PROGRAM PRG_05_Turret_Carriage
VAR
	R_TRIG_0: R_TRIG;
	R_TRIG_1: R_TRIG;
	F_TRIG_2: F_TRIG;
	F_TRIG_4: F_TRIG;
	RS_TriggerStopCCW: RS;
	R_TRIG_12: R_TRIG;
	RS_TriggerStopCW: RS;
	R_TRIG_15: R_TRIG;
	R_TRIG_18: R_TRIG;
	R_TRIG_19: R_TRIG;
	R_TRIG_20: R_TRIG;
	R_TRIG_21: R_TRIG;
	R_TRIG_22: R_TRIG;
	TOF_SwitchDelay: TOF;
	R_TRIG_23: R_TRIG;
	R_TRIG_24: R_TRIG;
	R_TRIG_25: R_TRIG;
	R_TRIG_26: R_TRIG;
	F_TRIG_0: F_TRIG;
	F_TRIG_1: F_TRIG;
END_VAR
VAR // added by the converter: edge detectors and wires of the graphical bodies
    _w1, _w2 : BOOL;
END_VAR

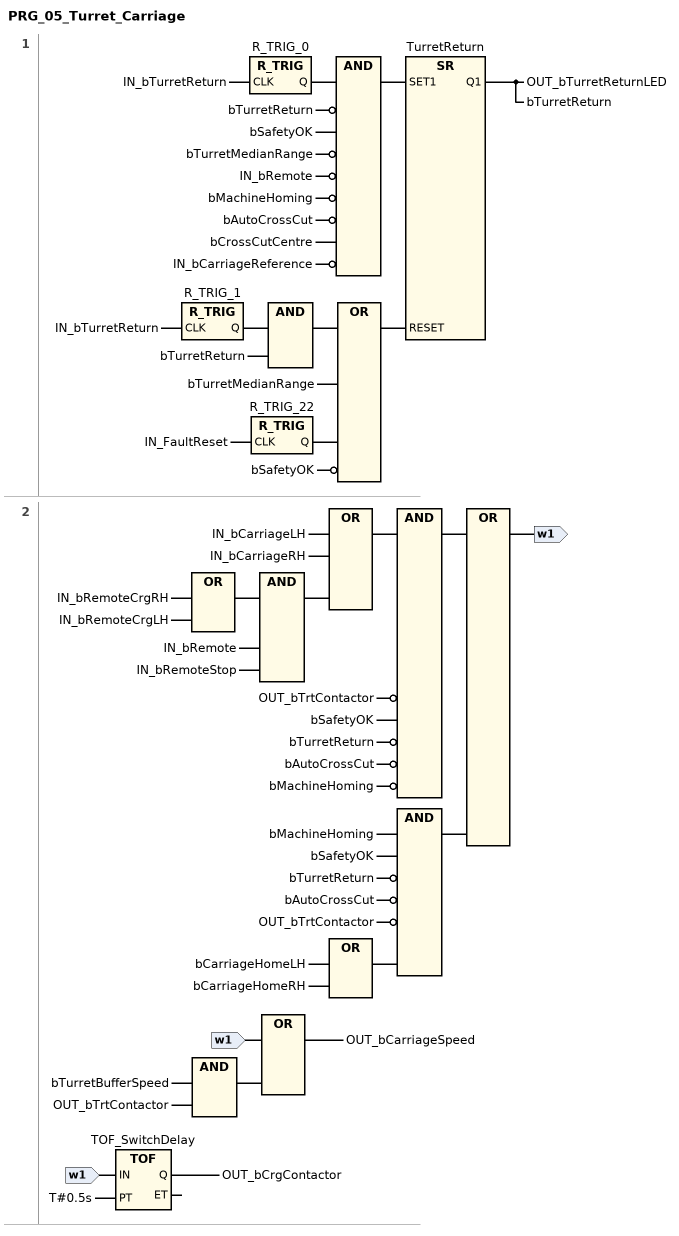
// NETWORK 1
R_TRIG_0(CLK := IN_bTurretReturn); // R_TRIG
R_TRIG_1(CLK := IN_bTurretReturn); // R_TRIG
R_TRIG_22(CLK := IN_FaultReset); // R_TRIG
TurretReturn(SET1 := R_TRIG_0.Q AND NOT bTurretReturn AND bSafetyOK AND NOT bTurretMedianRange AND NOT IN_bRemote AND NOT bMachineHoming AND NOT bAutoCrossCut AND bCrossCutCentre AND NOT IN_bCarriageReference, RESET := R_TRIG_1.Q AND bTurretReturn OR bTurretMedianRange OR R_TRIG_22.Q OR NOT bSafetyOK); // SR
OUT_bTurretReturnLED := TurretReturn.Q1;
bTurretReturn := TurretReturn.Q1;

// NETWORK 2
_w1 := (IN_bCarriageLH OR IN_bCarriageRH OR (IN_bRemoteCrgRH OR IN_bRemoteCrgLH) AND IN_bRemote AND IN_bRemoteStop) AND NOT OUT_bTrtContactor AND bSafetyOK AND NOT bTurretReturn AND NOT bAutoCrossCut AND NOT bMachineHoming OR bMachineHoming AND bSafetyOK AND NOT bTurretReturn AND NOT bAutoCrossCut AND NOT OUT_bTrtContactor AND (bCarriageHomeLH OR bCarriageHomeRH);
OUT_bCarriageSpeed := _w1 OR bTurretBufferSpeed AND OUT_bTrtContactor;
TOF_SwitchDelay(IN := _w1, PT := T#0.5s); // TOF
OUT_bCrgContactor := TOF_SwitchDelay.Q;

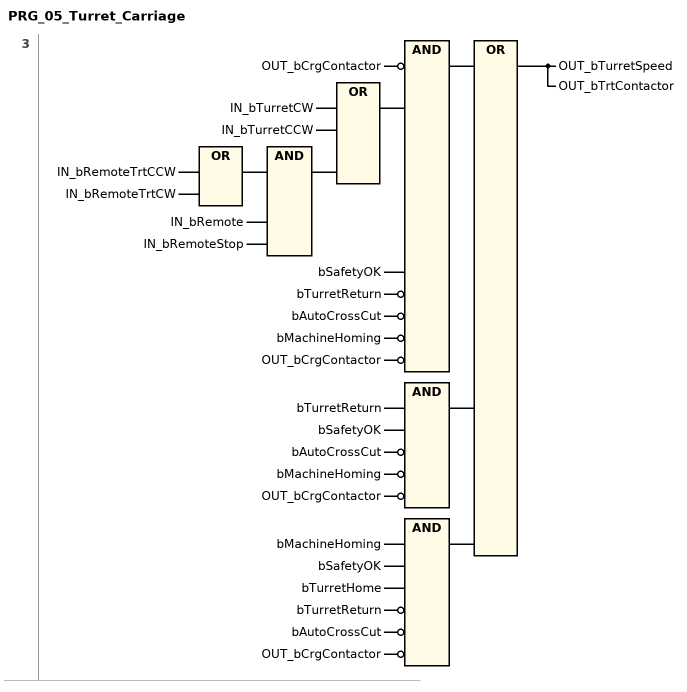
// NETWORK 3
_w2 := NOT OUT_bCrgContactor AND (IN_bTurretCW OR IN_bTurretCCW OR (IN_bRemoteTrtCCW OR IN_bRemoteTrtCW) AND IN_bRemote AND IN_bRemoteStop) AND bSafetyOK AND NOT bTurretReturn AND NOT bAutoCrossCut AND NOT bMachineHoming AND NOT OUT_bCrgContactor OR bTurretReturn AND bSafetyOK AND NOT bAutoCrossCut AND NOT bMachineHoming AND NOT OUT_bCrgContactor OR bMachineHoming AND bSafetyOK AND bTurretHome AND NOT bTurretReturn AND NOT bAutoCrossCut AND NOT OUT_bCrgContactor;
OUT_bTurretSpeed := _w2;
OUT_bTrtContactor := _w2;

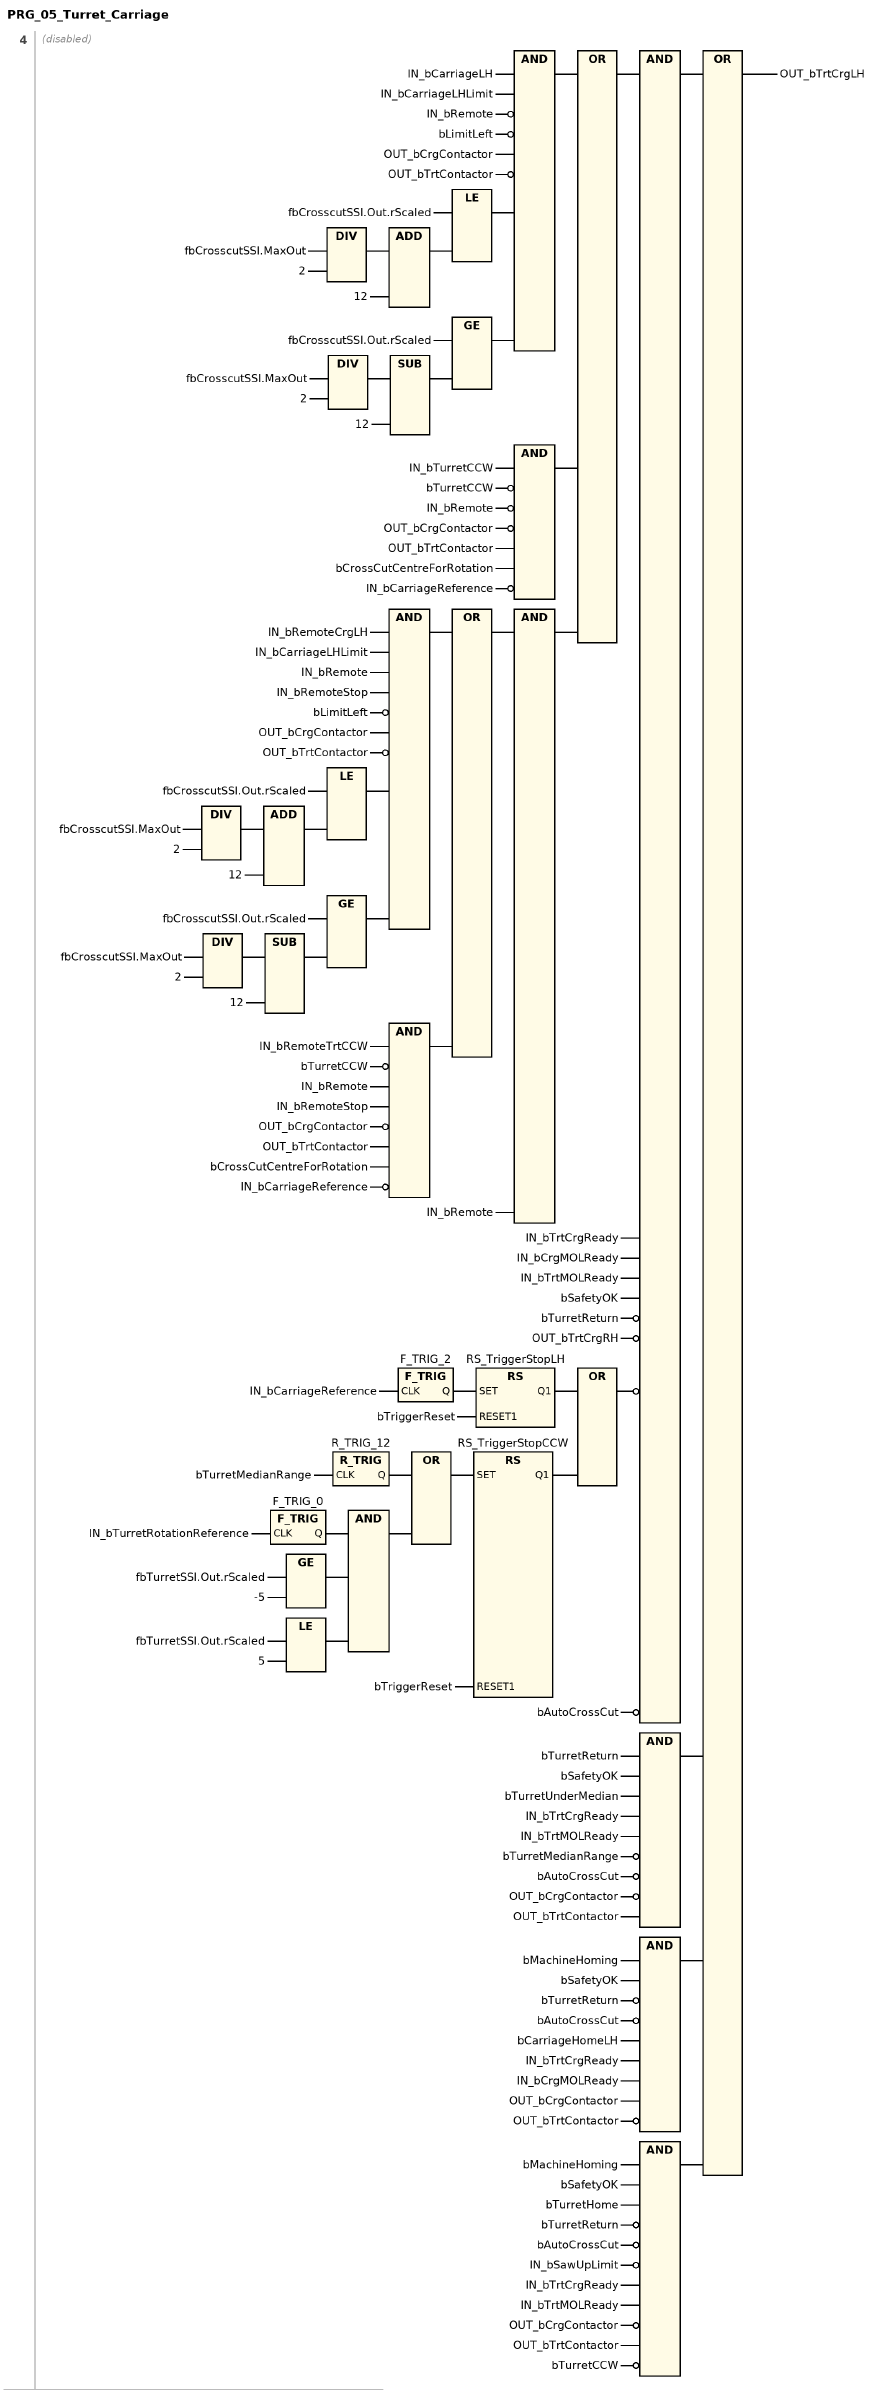
// NETWORK 4 (disabled)
// F_TRIG_2(CLK := IN_bCarriageReference); // F_TRIG
// RS_TriggerStopLH(SET := F_TRIG_2.Q, RESET1 := bTriggerReset); // RS
// R_TRIG_12(CLK := bTurretMedianRange); // R_TRIG
// F_TRIG_0(CLK := IN_bTurretRotationReference); // F_TRIG
// RS_TriggerStopCCW(SET := R_TRIG_12.Q OR F_TRIG_0.Q AND fbTurretSSI.Out.rScaled >= -5 AND fbTurretSSI.Out.rScaled <= 5, RESET1 := bTriggerReset); // RS
// OUT_bTrtCrgLH := (IN_bCarriageLH AND IN_bCarriageLHLimit AND NOT IN_bRemote AND NOT bLimitLeft AND OUT_bCrgContactor AND NOT OUT_bTrtContactor AND fbCrosscutSSI.Out.rScaled <= fbCrosscutSSI.MaxOut / 2 + 12 AND fbCrosscutSSI.Out.rScaled >= fbCrosscutSSI.MaxOut / 2 - 12 OR IN_bTurretCCW AND NOT bTurretCCW AND NOT IN_bRemote AND NOT OUT_bCrgContactor AND OUT_bTrtContactor AND bCrossCutCentreForRotation AND NOT IN_bCarriageReference OR (IN_bRemoteCrgLH AND IN_bCarriageLHLimit AND IN_bRemote AND IN_bRemoteStop AND NOT bLimitLeft AND OUT_bCrgContactor AND NOT OUT_bTrtContactor AND fbCrosscutSSI.Out.rScaled <= fbCrosscutSSI.MaxOut / 2 + 12 AND fbCrosscutSSI.Out.rScaled >= fbCrosscutSSI.MaxOut / 2 - 12 OR IN_bRemoteTrtCCW AND NOT bTurretCCW AND IN_bRemote AND IN_bRemoteStop AND NOT OUT_bCrgContactor AND OUT_bTrtContactor AND bCrossCutCentreForRotation AND NOT IN_bCarriageReference) AND IN_bRemote) AND IN_bTrtCrgReady AND IN_bCrgMOLReady AND IN_bTrtMOLReady AND bSafetyOK AND NOT bTurretReturn AND NOT OUT_bTrtCrgRH AND NOT (RS_TriggerStopLH.Q1 OR RS_TriggerStopCCW.Q1) AND NOT bAutoCrossCut OR bTurretReturn AND bSafetyOK AND bTurretUnderMedian AND IN_bTrtCrgReady AND IN_bTrtMOLReady AND NOT bTurretMedianRange AND NOT bAutoCrossCut AND NOT OUT_bCrgContactor AND OUT_bTrtContactor OR bMachineHoming AND bSafetyOK AND NOT bTurretReturn AND NOT bAutoCrossCut AND bCarriageHomeLH AND IN_bTrtCrgReady AND IN_bCrgMOLReady AND OUT_bCrgContactor AND NOT OUT_bTrtContactor OR bMachineHoming AND bSafetyOK AND bTurretHome AND NOT bTurretReturn AND NOT bAutoCrossCut AND NOT IN_bSawUpLimit AND IN_bTrtCrgReady AND IN_bTrtMOLReady AND NOT OUT_bCrgContactor AND OUT_bTrtContactor AND NOT bTurretCCW;

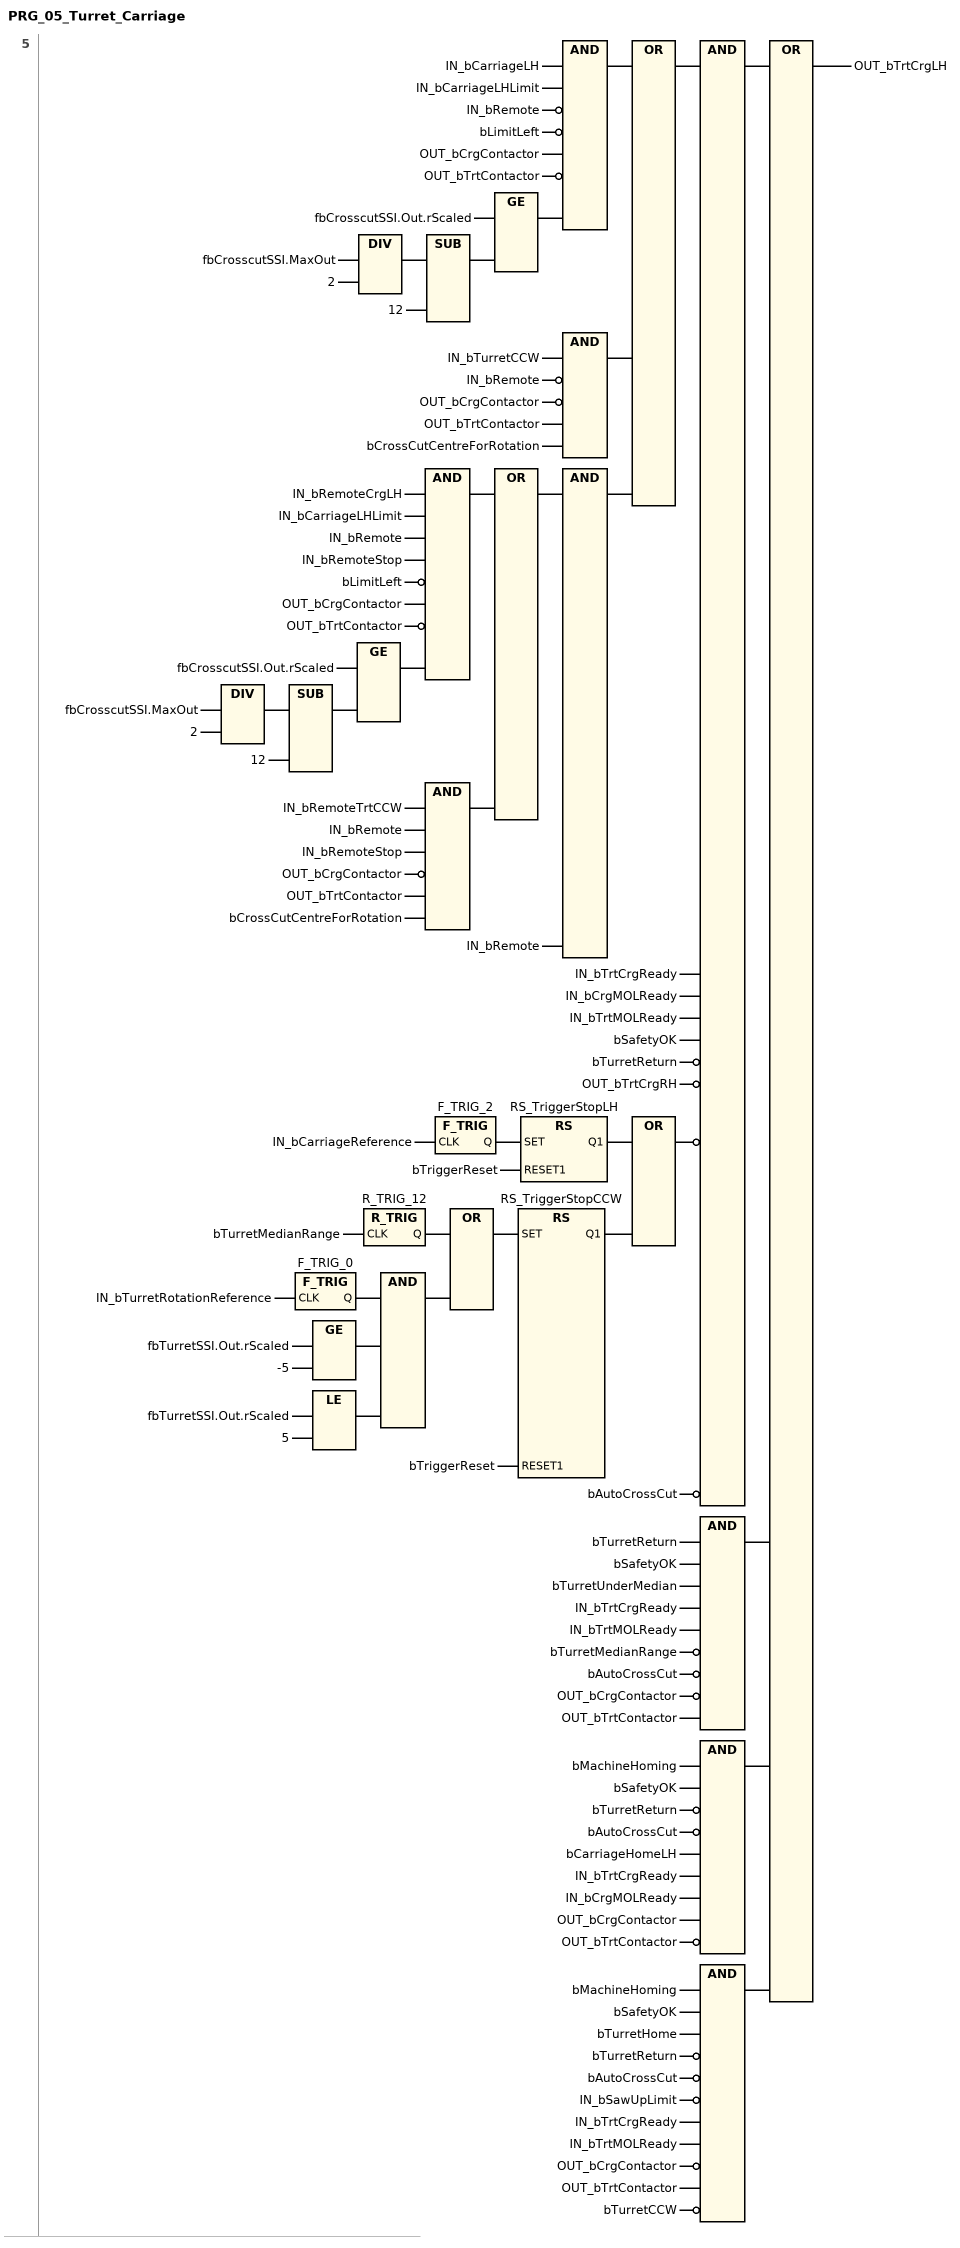
// NETWORK 5
F_TRIG_2(CLK := IN_bCarriageReference); // F_TRIG
RS_TriggerStopLH(SET := F_TRIG_2.Q, RESET1 := bTriggerReset); // RS
R_TRIG_12(CLK := bTurretMedianRange); // R_TRIG
F_TRIG_0(CLK := IN_bTurretRotationReference); // F_TRIG
RS_TriggerStopCCW(SET := R_TRIG_12.Q OR F_TRIG_0.Q AND fbTurretSSI.Out.rScaled >= -5 AND fbTurretSSI.Out.rScaled <= 5, RESET1 := bTriggerReset); // RS
OUT_bTrtCrgLH := (IN_bCarriageLH AND IN_bCarriageLHLimit AND NOT IN_bRemote AND NOT bLimitLeft AND OUT_bCrgContactor AND NOT OUT_bTrtContactor AND fbCrosscutSSI.Out.rScaled >= fbCrosscutSSI.MaxOut / 2 - 12 OR IN_bTurretCCW AND NOT IN_bRemote AND NOT OUT_bCrgContactor AND OUT_bTrtContactor AND bCrossCutCentreForRotation OR (IN_bRemoteCrgLH AND IN_bCarriageLHLimit AND IN_bRemote AND IN_bRemoteStop AND NOT bLimitLeft AND OUT_bCrgContactor AND NOT OUT_bTrtContactor AND fbCrosscutSSI.Out.rScaled >= fbCrosscutSSI.MaxOut / 2 - 12 OR IN_bRemoteTrtCCW AND IN_bRemote AND IN_bRemoteStop AND NOT OUT_bCrgContactor AND OUT_bTrtContactor AND bCrossCutCentreForRotation) AND IN_bRemote) AND IN_bTrtCrgReady AND IN_bCrgMOLReady AND IN_bTrtMOLReady AND bSafetyOK AND NOT bTurretReturn AND NOT OUT_bTrtCrgRH AND NOT (RS_TriggerStopLH.Q1 OR RS_TriggerStopCCW.Q1) AND NOT bAutoCrossCut OR bTurretReturn AND bSafetyOK AND bTurretUnderMedian AND IN_bTrtCrgReady AND IN_bTrtMOLReady AND NOT bTurretMedianRange AND NOT bAutoCrossCut AND NOT OUT_bCrgContactor AND OUT_bTrtContactor OR bMachineHoming AND bSafetyOK AND NOT bTurretReturn AND NOT bAutoCrossCut AND bCarriageHomeLH AND IN_bTrtCrgReady AND IN_bCrgMOLReady AND OUT_bCrgContactor AND NOT OUT_bTrtContactor OR bMachineHoming AND bSafetyOK AND bTurretHome AND NOT bTurretReturn AND NOT bAutoCrossCut AND NOT IN_bSawUpLimit AND IN_bTrtCrgReady AND IN_bTrtMOLReady AND NOT OUT_bCrgContactor AND OUT_bTrtContactor AND NOT bTurretCCW;

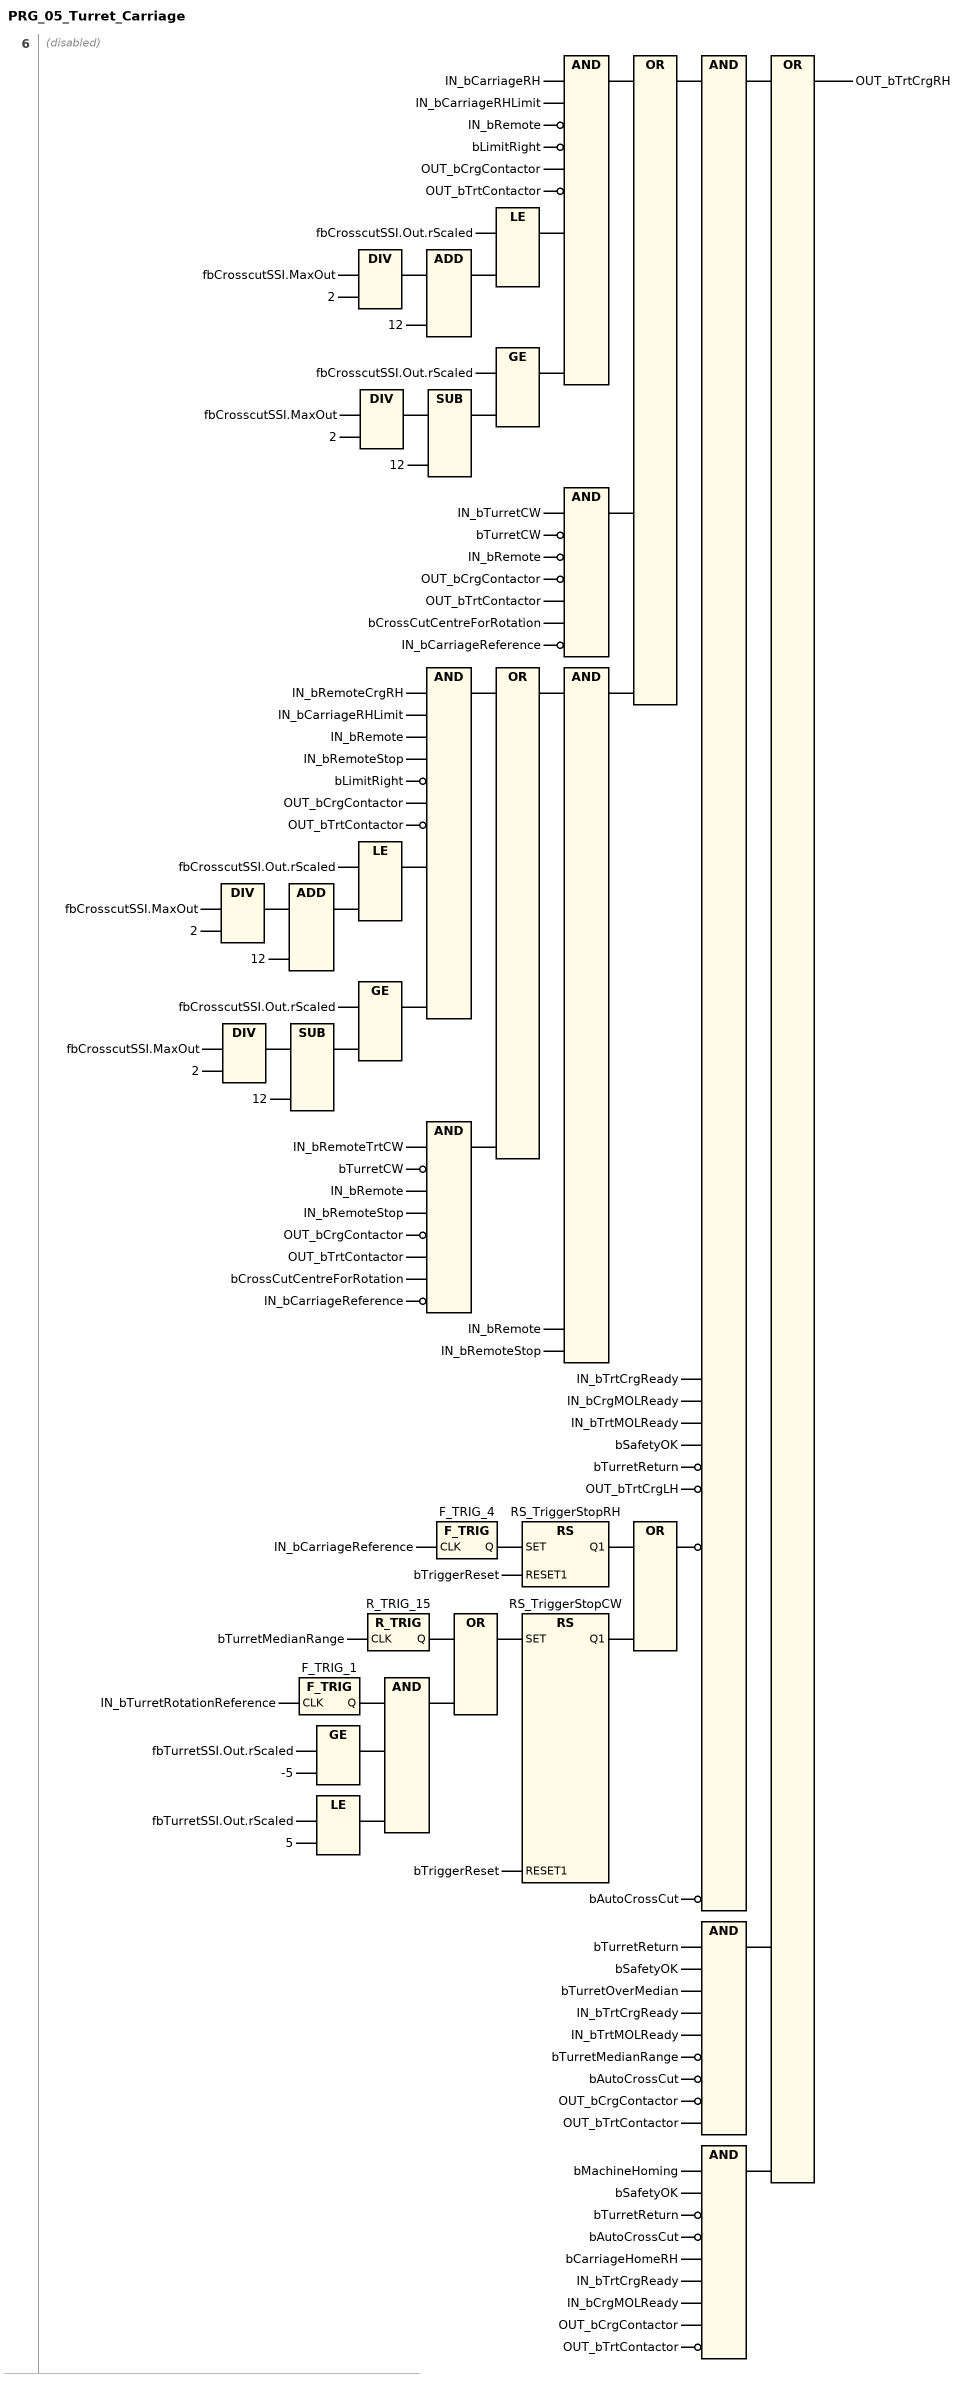
// NETWORK 6 (disabled)
// F_TRIG_4(CLK := IN_bCarriageReference); // F_TRIG
// RS_TriggerStopRH(SET := F_TRIG_4.Q, RESET1 := bTriggerReset); // RS
// R_TRIG_15(CLK := bTurretMedianRange); // R_TRIG
// F_TRIG_1(CLK := IN_bTurretRotationReference); // F_TRIG
// RS_TriggerStopCW(SET := R_TRIG_15.Q OR F_TRIG_1.Q AND fbTurretSSI.Out.rScaled >= -5 AND fbTurretSSI.Out.rScaled <= 5, RESET1 := bTriggerReset); // RS
// OUT_bTrtCrgRH := (IN_bCarriageRH AND IN_bCarriageRHLimit AND NOT IN_bRemote AND NOT bLimitRight AND OUT_bCrgContactor AND NOT OUT_bTrtContactor AND fbCrosscutSSI.Out.rScaled <= fbCrosscutSSI.MaxOut / 2 + 12 AND fbCrosscutSSI.Out.rScaled >= fbCrosscutSSI.MaxOut / 2 - 12 OR IN_bTurretCW AND NOT bTurretCW AND NOT IN_bRemote AND NOT OUT_bCrgContactor AND OUT_bTrtContactor AND bCrossCutCentreForRotation AND NOT IN_bCarriageReference OR (IN_bRemoteCrgRH AND IN_bCarriageRHLimit AND IN_bRemote AND IN_bRemoteStop AND NOT bLimitRight AND OUT_bCrgContactor AND NOT OUT_bTrtContactor AND fbCrosscutSSI.Out.rScaled <= fbCrosscutSSI.MaxOut / 2 + 12 AND fbCrosscutSSI.Out.rScaled >= fbCrosscutSSI.MaxOut / 2 - 12 OR IN_bRemoteTrtCW AND NOT bTurretCW AND IN_bRemote AND IN_bRemoteStop AND NOT OUT_bCrgContactor AND OUT_bTrtContactor AND bCrossCutCentreForRotation AND NOT IN_bCarriageReference) AND IN_bRemote AND IN_bRemoteStop) AND IN_bTrtCrgReady AND IN_bCrgMOLReady AND IN_bTrtMOLReady AND bSafetyOK AND NOT bTurretReturn AND NOT OUT_bTrtCrgLH AND NOT (RS_TriggerStopRH.Q1 OR RS_TriggerStopCW.Q1) AND NOT bAutoCrossCut OR bTurretReturn AND bSafetyOK AND bTurretOverMedian AND IN_bTrtCrgReady AND IN_bTrtMOLReady AND NOT bTurretMedianRange AND NOT bAutoCrossCut AND NOT OUT_bCrgContactor AND OUT_bTrtContactor OR bMachineHoming AND bSafetyOK AND NOT bTurretReturn AND NOT bAutoCrossCut AND bCarriageHomeRH AND IN_bTrtCrgReady AND IN_bCrgMOLReady AND OUT_bCrgContactor AND NOT OUT_bTrtContactor;

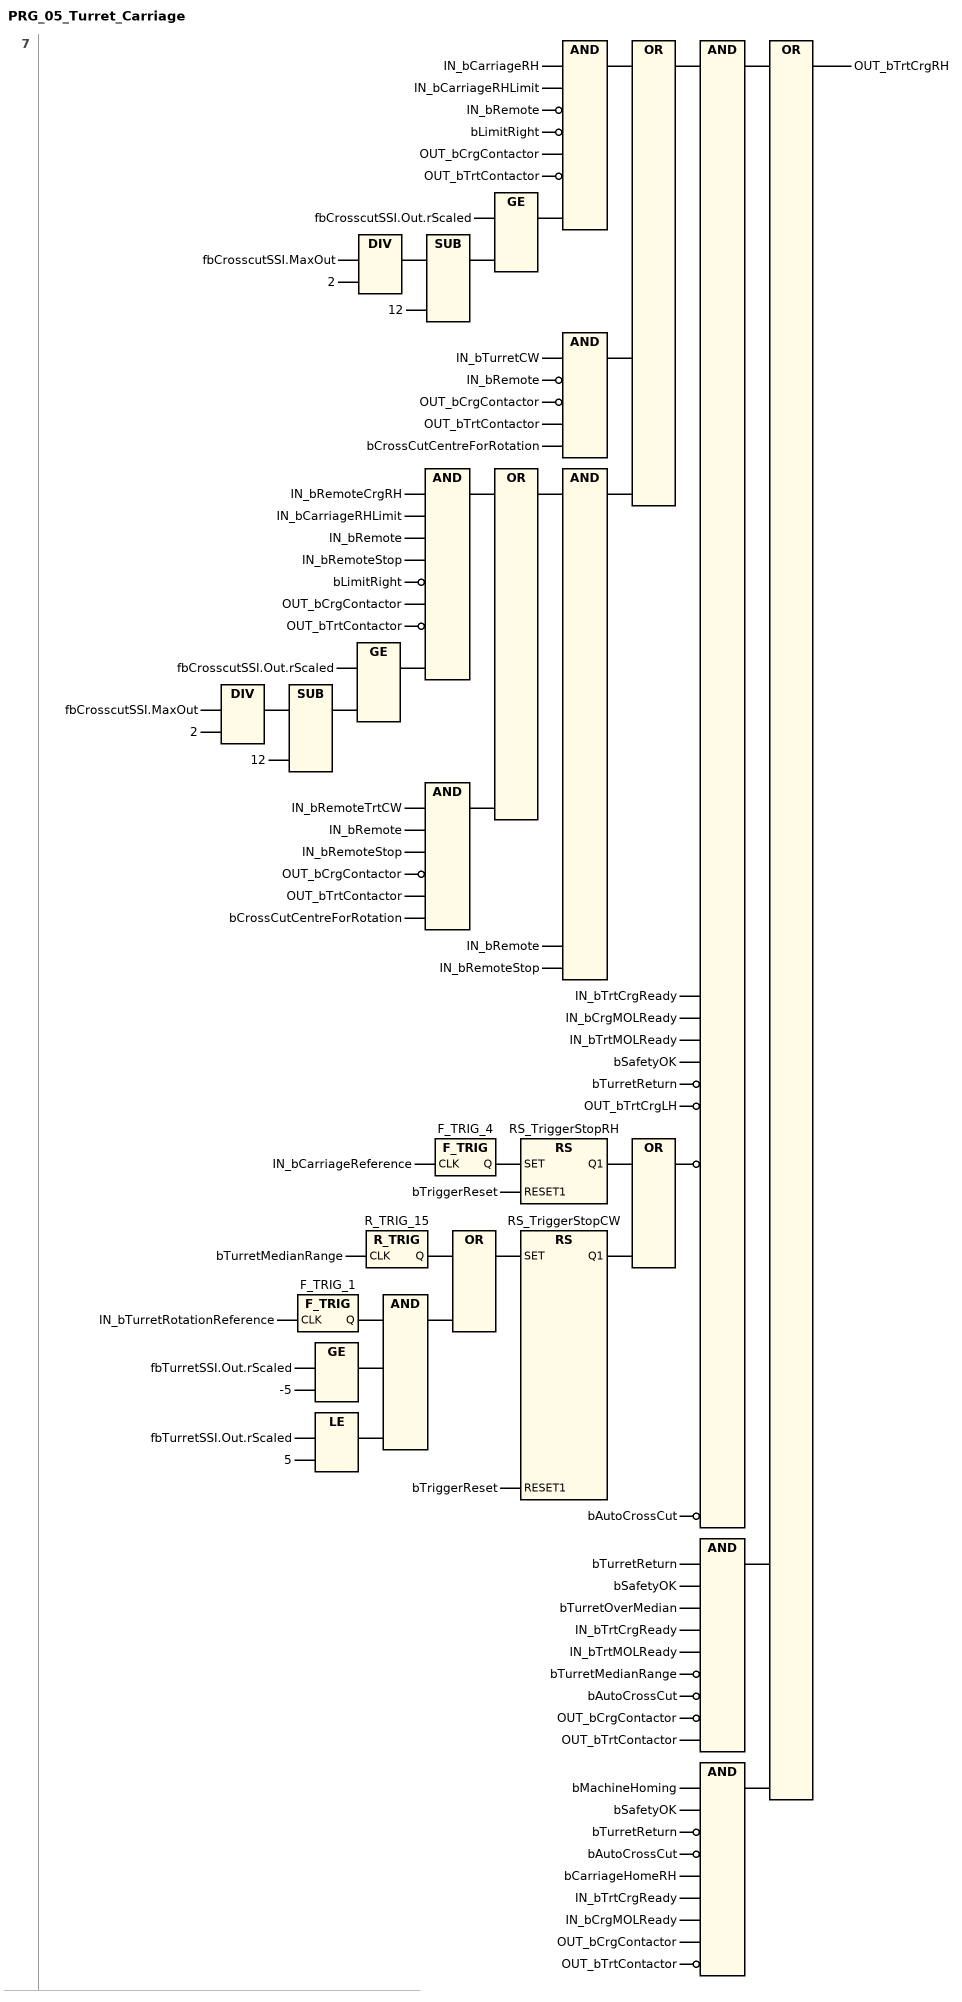
// NETWORK 7
F_TRIG_4(CLK := IN_bCarriageReference); // F_TRIG
RS_TriggerStopRH(SET := F_TRIG_4.Q, RESET1 := bTriggerReset); // RS
R_TRIG_15(CLK := bTurretMedianRange); // R_TRIG
F_TRIG_1(CLK := IN_bTurretRotationReference); // F_TRIG
RS_TriggerStopCW(SET := R_TRIG_15.Q OR F_TRIG_1.Q AND fbTurretSSI.Out.rScaled >= -5 AND fbTurretSSI.Out.rScaled <= 5, RESET1 := bTriggerReset); // RS
OUT_bTrtCrgRH := (IN_bCarriageRH AND IN_bCarriageRHLimit AND NOT IN_bRemote AND NOT bLimitRight AND OUT_bCrgContactor AND NOT OUT_bTrtContactor AND fbCrosscutSSI.Out.rScaled >= fbCrosscutSSI.MaxOut / 2 - 12 OR IN_bTurretCW AND NOT IN_bRemote AND NOT OUT_bCrgContactor AND OUT_bTrtContactor AND bCrossCutCentreForRotation OR (IN_bRemoteCrgRH AND IN_bCarriageRHLimit AND IN_bRemote AND IN_bRemoteStop AND NOT bLimitRight AND OUT_bCrgContactor AND NOT OUT_bTrtContactor AND fbCrosscutSSI.Out.rScaled >= fbCrosscutSSI.MaxOut / 2 - 12 OR IN_bRemoteTrtCW AND IN_bRemote AND IN_bRemoteStop AND NOT OUT_bCrgContactor AND OUT_bTrtContactor AND bCrossCutCentreForRotation) AND IN_bRemote AND IN_bRemoteStop) AND IN_bTrtCrgReady AND IN_bCrgMOLReady AND IN_bTrtMOLReady AND bSafetyOK AND NOT bTurretReturn AND NOT OUT_bTrtCrgLH AND NOT (RS_TriggerStopRH.Q1 OR RS_TriggerStopCW.Q1) AND NOT bAutoCrossCut OR bTurretReturn AND bSafetyOK AND bTurretOverMedian AND IN_bTrtCrgReady AND IN_bTrtMOLReady AND NOT bTurretMedianRange AND NOT bAutoCrossCut AND NOT OUT_bCrgContactor AND OUT_bTrtContactor OR bMachineHoming AND bSafetyOK AND NOT bTurretReturn AND NOT bAutoCrossCut AND bCarriageHomeRH AND IN_bTrtCrgReady AND IN_bCrgMOLReady AND OUT_bCrgContactor AND NOT OUT_bTrtContactor;

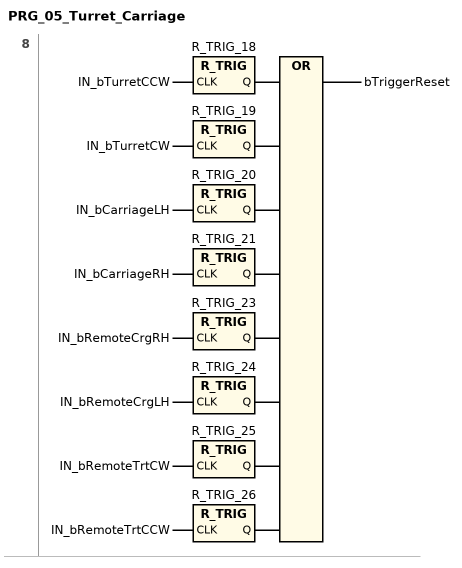
// NETWORK 8
R_TRIG_18(CLK := IN_bTurretCCW); // R_TRIG
R_TRIG_19(CLK := IN_bTurretCW); // R_TRIG
R_TRIG_20(CLK := IN_bCarriageLH); // R_TRIG
R_TRIG_21(CLK := IN_bCarriageRH); // R_TRIG
R_TRIG_23(CLK := IN_bRemoteCrgRH); // R_TRIG
R_TRIG_24(CLK := IN_bRemoteCrgLH); // R_TRIG
R_TRIG_25(CLK := IN_bRemoteTrtCW); // R_TRIG
R_TRIG_26(CLK := IN_bRemoteTrtCCW); // R_TRIG
bTriggerReset := R_TRIG_18.Q OR R_TRIG_19.Q OR R_TRIG_20.Q OR R_TRIG_21.Q OR R_TRIG_23.Q OR R_TRIG_24.Q OR R_TRIG_25.Q OR R_TRIG_26.Q;

END_PROGRAM

(* stored: Version 1.1.0.1, ProductVersion 3.1.4024.12
   POU PRG_05_Turret_Carriage: Id {70aa8ac8-a439-4b47-9352-f3d2b02948a6}, SpecialFunc None *)
